// Mitsubishi GX Works2 project: FBD_op_matematicas   PLC: Q03UDV

// task Task_01 (event TRUE, interval 0, priority 31): POU_01

PROGRAM POU_01
(* structured ladder/FBD written out as ST: instructions are called as NAME(EN, inputs, outputs); _pN, _eN, _tN stand for wires *)
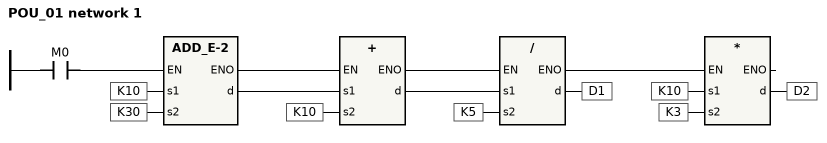
(* network 1 *)
_e2 := ADD_E(M0, K10, K30, _t1);
_e4 := +(_e2, _t1, K10, _t3);
_e5 := /(_e4, _t3, K5, D1);
*(_e5, K10, K3, D2);
END_PROGRAM
